INTERFACE I_Axis

METHOD AbsMove : BOOL
VAR_INPUT
	// 目標位置
	_Position : LREAL;
	// 移動速度
	_Velocity : LREAL := 0;
END_VAR
END_METHOD

PROPERTY Buzy : bool
GET
END_GET
END_PROPERTY

PROPERTY Done : bool
GET
END_GET
END_PROPERTY

PROPERTY Error : bool
GET
END_GET
END_PROPERTY

METHOD Homing : BOOL
VAR_INPUT
END_VAR
END_METHOD

METHOD PowerOff : BOOL
VAR_INPUT
END_VAR
END_METHOD

METHOD PowerOn : BOOL
VAR_INPUT
END_VAR
END_METHOD

METHOD RelMove : BOOL
VAR_INPUT
	// 目標距離
	_Position : LREAL;
	
	// 移動速度
	_Velocity : LREAL := 0;
END_VAR
END_METHOD

METHOD SetLimit : BOOL
VAR_INPUT
END_VAR
END_METHOD

METHOD Stop : BOOL
VAR_INPUT
END_VAR
END_METHOD

END_INTERFACE

(* stored: Version 1.1.0.1, ProductVersion 3.1.4024.15
   Itf I_Axis: Id {a2f5afd8-61ff-4878-816a-4ca5499ac4b6}
   Method AbsMove: Id {b4dc91c9-c383-4703-bbd3-000f8b7fe4f3}
   Property Buzy: Id {13ff5930-4189-47aa-a91b-2626629d1e7c}
   Get Get: Id {e52d5f37-31e3-4df1-85fc-b2c530c5e1ff}
   Property Done: Id {7675a719-25c9-49a8-aa5e-6aeb46792787}
   Get Get: Id {4ee689db-aabe-43cd-a417-196e57257012}
   Property Error: Id {80875dbb-22b0-4636-917e-070193a4c627}
   Get Get: Id {7d38247e-4677-4f10-a029-7bda424a6f44}
   Method Homing: Id {eec6ceac-2926-44c3-8892-6d7043d7a6d5}
   Method PowerOff: Id {e8b45e22-e631-4a5d-b7ba-8466121012ec}
   Method PowerOn: Id {409dea29-ddcf-40de-8413-2c694b940eaf}
   Method RelMove: Id {eb098bf2-47a0-4747-9431-92eeba89ae7e}
   Method SetLimit: Id {42cd9e6b-fcbd-4a85-b878-08cbb0879eeb}
   Method Stop: Id {f6d44283-9ee6-4ff4-b3e7-b3991147eb26} *)
